// SIMATIC STEP 7 (V5.x) project GYDS201808
// CPU: CPU 315-2 PN/DP
// station: P_ADR_BUS
// station: 硬件
// station: SIMATIC 300(1)
// program: S7 程序(2)

DATA_BLOCK DB 1
VERSION : 0.1
  STRUCT
   TEMP_TAG1 : BOOL ;	//TEMP_TAG1
  END_STRUCT ;	
BEGIN
END_DATA_BLOCK

DATA_BLOCK DB 2
VERSION : 0.1
  STRUCT
   DB_VAR : BOOL ;	//临时占位符变量
  END_STRUCT ;	
BEGIN
END_DATA_BLOCK

DATA_BLOCK DB 3
VERSION : 0.1
  STRUCT
   DB_VAR : INT ;	//临时占位符变量
  END_STRUCT ;	
BEGIN
END_DATA_BLOCK

DATA_BLOCK DB 4
VERSION : 0.1
  STRUCT
   DB_VAR : INT ;	//临时占位符变量
  END_STRUCT ;	
BEGIN
END_DATA_BLOCK

DATA_BLOCK DB 5
VERSION : 0.1
  STRUCT
   DB_VAR : INT ;	//临时占位符变量
  END_STRUCT ;	
BEGIN
END_DATA_BLOCK

DATA_BLOCK DB 6
VERSION : 0.1
  STRUCT
   DB_VAR : INT ;	//临时占位符变量
  END_STRUCT ;	
BEGIN
END_DATA_BLOCK

DATA_BLOCK DB 7
VERSION : 0.1
  STRUCT
   DB_VAR : BOOL ;	//临时占位符变量
  END_STRUCT ;	
BEGIN
END_DATA_BLOCK

DATA_BLOCK DB 8
VERSION : 0.1
  STRUCT
   DB_VAR : BOOL ;	//临时占位符变量
  END_STRUCT ;	
BEGIN
END_DATA_BLOCK

DATA_BLOCK DB 9
VERSION : 0.1
  STRUCT
   DB_VAR : INT ;	//临时占位符变量
  END_STRUCT ;	
BEGIN
END_DATA_BLOCK

DATA_BLOCK DB 10
VERSION : 0.1
  STRUCT
   DB_VAR : INT ;	//临时占位符变量
  END_STRUCT ;	
BEGIN
END_DATA_BLOCK

DATA_BLOCK DB 11
VERSION : 0.1
  STRUCT
   DB_VAR : INT  := 2;	//临时占位符变量
  END_STRUCT ;	
BEGIN
END_DATA_BLOCK

DATA_BLOCK DB 20
VERSION : 0.1
  STRUCT
   DB_VAR : INT ;	//临时占位符变量
  END_STRUCT ;	
BEGIN
END_DATA_BLOCK

ORGANIZATION_BLOCK OB 1
TITLE = "Main Program Sweep (Cycle)"
VERSION : 0.1
VAR_TEMP
  OB1_EV_CLASS : BYTE ;	//Bits 0-3 = 1 (Coming event), Bits 4-7 = 1 (Event class 1)
  OB1_SCAN_1 : BYTE ;	//1 (Cold restart scan 1 of OB 1), 3 (Scan 2-n of OB 1)
  OB1_PRIORITY : BYTE ;	//Priority of OB Execution
  OB1_OB_NUMBR : BYTE ;	//1 (Organization block 1, OB1)
  OB1_RESERVED_1 : BYTE ;	//Reserved for system
  OB1_RESERVED_2 : BYTE ;	//Reserved for system
  OB1_PREV_CYCLE : INT ;	//Cycle time of previous OB1 scan (milliseconds)
  OB1_MIN_CYCLE : INT ;	//Minimum cycle time of OB1 (milliseconds)
  OB1_MAX_CYCLE : INT ;	//Maximum cycle time of OB1 (milliseconds)
  OB1_DATE_TIME : DATE_AND_TIME ;	//Date and time OB1 started
END_VAR
BEGIN
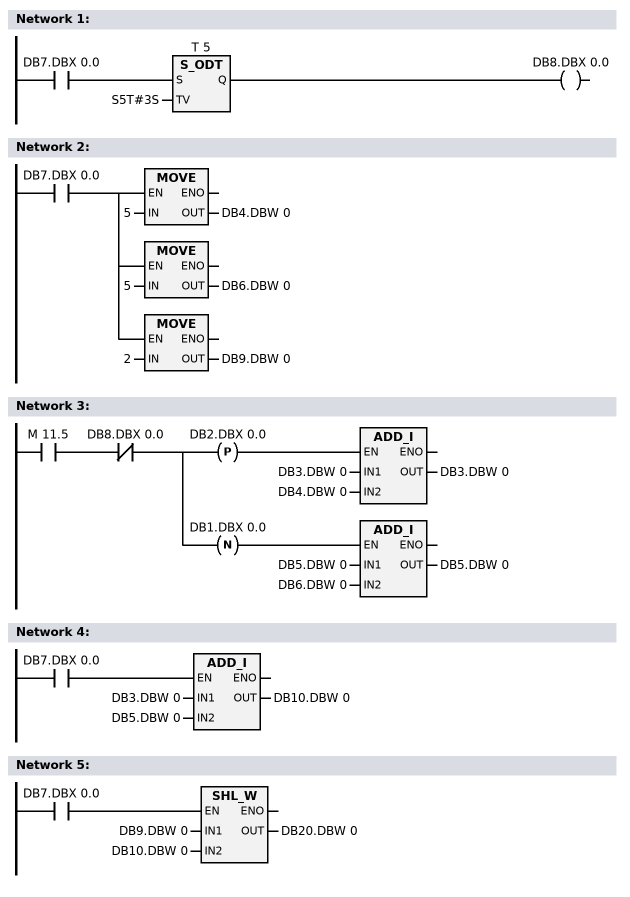
NETWORK
TITLE =
      A     DB7.DBX 0.0;
      L     S5T#3S;
      SD    T 5;
      NOP   0;
      NOP   0;
      NOP   0;
      A     T 5;
      =     DB8.DBX 0.0;
NETWORK
TITLE =
      A     DB7.DBX 0.0;
      =     L 20.0;
      A     L 20.0;
      JNB   _001;
      L     5;
      T     DB4.DBW 0;
_001: NOP   0;
      A     L 20.0;
      JNB   _002;
      L     5;
      T     DB6.DBW 0;
_002: NOP   0;
      A     L 20.0;
      JNB   _003;
      L     2;
      T     DB9.DBW 0;
_003: NOP   0;
NETWORK
TITLE =
      A     M 11.5;
      AN    DB8.DBX 0.0;
      =     L 20.0;
      A     L 20.0;
      FP    DB2.DBX 0.0;
      JNB   _004;
      L     DB3.DBW 0;
      L     DB4.DBW 0;
      +I;
      T     DB3.DBW 0;
_004: NOP   0;
      A     L 20.0;
      FN    DB1.DBX 0.0;
      JNB   _005;
      L     DB5.DBW 0;
      L     DB6.DBW 0;
      +I;
      T     DB5.DBW 0;
_005: NOP   0;
NETWORK
TITLE =
      A     DB7.DBX 0.0;
      JNB   _006;
      L     DB3.DBW 0;
      L     DB5.DBW 0;
      +I;
      T     DB10.DBW 0;
_006: NOP   0;
NETWORK
TITLE =
      A     DB7.DBX 0.0;
      JNB   _007;
      L     DB9.DBW 0;
      L     DB10.DBW 0;
      SLW;
      T     DB20.DBW 0;
_007: NOP   0;
END_ORGANIZATION_BLOCK
